ADAPTER SetParams1Word (* Adapter Interface *)
  (* Standard: 61499-1 *)
  (* Version 1.0, 2021-10-04, dorofeev *)
  (* Compiler header: package fb.test; *)
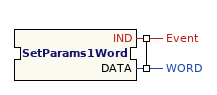
  EVENT_OUTPUT
    IND WITH DATA; (* Indication from Plug *)
  END_EVENT
  VAR_OUTPUT
    DATA : WORD; (* Indication Data from Plug *)
  END_VAR
  SERVICE PLUG/SOCKET (* Adapter Interface *)
    SEQUENCE normal_operation
      PLUG.IND(DATA=1) -> SOCKET.IND(DATA=1);
    END_SEQUENCE
    SEQUENCE indication_response
    END_SEQUENCE
  END_SERVICE
END_ADAPTER
